// TIA Portal V20 export
DATA_BLOCK "Temperatur_DB"   // DB109
// stored: InstanceOfName Temperatur, InstanceOfType FB
"Temperatur"
   // VAR_INPUT
   //    Temp_Set : Real;
   //    Level : Real;
   // END_VAR
   // VAR_OUTPUT
   //    Temp_Current : Real;
   //    TempCurrent_RAW : Int;
   // END_VAR
   // VAR
   //    Temp_amb : Real;
   //    c : Real;
   //    HeatOutput : Real;
   //    LossFactor : Real;
   //    "dt" : Real;
   // END_VAR
BEGIN
END_DATA_BLOCK
